FUNCTION_BLOCK FB_Startup
VAR_INPUT
END_VAR
VAR_OUTPUT
END_VAR
VAR
	timer1 : TON;
	timer2 : TON;
	timer3 : TON;
	timer4 : TON;
	timer5 : TON;
	timer6 : TON;
	timer7 : TON;
	timer14: INT;
END_VAR

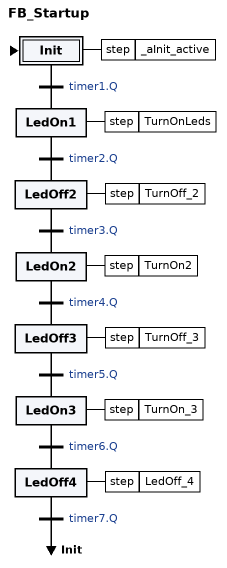
INITIAL_STEP Init:
    _aInit_active(N);  // step action
END_STEP
TRANSITION FROM Init TO LedOn1
    := timer1.Q;
END_TRANSITION
STEP LedOn1:
    TurnOnLeds(N);  // step action
END_STEP
TRANSITION FROM LedOn1 TO LedOff2
    := timer2.Q;
END_TRANSITION
STEP LedOff2:
    TurnOff_2(N);  // step action
END_STEP
TRANSITION FROM LedOff2 TO LedOn2
    := timer3.Q;
END_TRANSITION
STEP LedOn2:
    TurnOn2(N);  // step action
END_STEP
TRANSITION FROM LedOn2 TO LedOff3
    := timer4.Q;
END_TRANSITION
STEP LedOff3:
    TurnOff_3(N);  // step action
END_STEP
TRANSITION FROM LedOff3 TO LedOn3
    := timer5.Q;
END_TRANSITION
STEP LedOn3:
    TurnOn_3(N);  // step action
END_STEP
TRANSITION FROM LedOn3 TO LedOff4
    := timer6.Q;
END_TRANSITION
STEP LedOff4:
    LedOff_4(N);  // step action
END_STEP
TRANSITION FROM LedOff4 TO Init
    := timer7.Q;
END_TRANSITION

ACTION _aInit_active:
timer1(IN := TRUE, PT := T#1S);
timer2(IN := FALSE, PT := T#1S);
timer3(IN := FALSE, PT := T#1S);
timer4(IN := FALSE, PT := T#1S);
timer5(IN := FALSE, PT := T#1S);
timer6(IN := FALSE, PT := T#1S);
timer7(IN := FALSE, PT := T#1S);
AllLEDsTrigger(FALSE);
END_ACTION

METHOD AllLEDsTrigger : BOOL
VAR_INPUT
	OnOff : BOOL; // OnOff - Turn off, True - Turn On
END_VAR
GVL.LED_Comm_Fault := OnOff;
GVL.LED_EE_Grip := OnOff;
GVL.LED_EE_Ungrip := OnOff;
GVL.LED_EMG_STOP := OnOff;
GVL.LED_J1_CCW := OnOff;
GVL.LED_J1_CW := OnOff;
GVL.LED_J2_CCW := OnOff;
GVL.LED_J2_CW := OnOff;
GVL.LED_J3_CCW := OnOff;
GVL.LED_Record_Delay := OnOff;
GVL.LED_Record_Pos := OnOff;
GVL.LED_Reset := OnOff;
GVL.LED_Start_Pause := OnOff;
GVL.LED_Warning := OnOff;
END_METHOD

ACTION LedOff_4:
timer1(IN := FALSE, PT := T#1S);
timer2(IN := FALSE, PT := T#1S);
timer3(IN := FALSE, PT := T#1S);
timer4(IN := FALSE, PT := T#1S);
timer5(IN := FALSE, PT := T#1S);
timer6(IN := FALSE, PT := T#1S);
timer7(IN := TRUE, PT := T#1S);
AllLEDsTrigger(FALSE);
END_ACTION

ACTION TurnOff_2:
timer1(IN := FALSE, PT := T#1S);
timer2(IN := FALSE, PT := T#1S);
timer3(IN := TRUE, PT := T#1S);
timer4(IN := FALSE, PT := T#1S);
timer5(IN := FALSE, PT := T#1S);
timer6(IN := FALSE, PT := T#1S);
timer7(IN := FALSE, PT := T#1S);
AllLEDsTrigger(FALSE);
END_ACTION

ACTION TurnOff_3:
timer1(IN := FALSE, PT := T#1S);
timer2(IN := FALSE, PT := T#1S);
timer3(IN := FALSE, PT := T#1S);
timer4(IN := FALSE, PT := T#1S);
timer5(IN := TRUE, PT := T#1S);
timer6(IN := FALSE, PT := T#1S);
timer7(IN := FALSE, PT := T#1S);
AllLEDsTrigger(FALSE);
END_ACTION

ACTION TurnOn_3:
timer1(IN := FALSE, PT := T#1S);
timer2(IN := FALSE, PT := T#1S);
timer3(IN := FALSE, PT := T#1S);
timer4(IN := FALSE, PT := T#1S);
timer5(IN := FALSE, PT := T#1S);
timer6(IN := TRUE, PT := T#1S);
timer7(IN := FALSE, PT := T#1S);
AllLEDsTrigger(TRUE);
END_ACTION

ACTION TurnOn2:
timer1(IN := FALSE, PT := T#1S);
timer2(IN := FALSE, PT := T#1S);
timer3(IN := FALSE, PT := T#1S);
timer4(IN := TRUE, PT := T#1S);
timer5(IN := FALSE, PT := T#1S);
timer6(IN := FALSE, PT := T#1S);
timer7(IN := FALSE, PT := T#1S);
AllLEDsTrigger(TRUE);
END_ACTION

ACTION TurnOnLeds:
timer1(IN := FALSE, PT := T#1S);
timer2(IN := TRUE, PT := T#1S);
timer3(IN := FALSE, PT := T#1S);
timer4(IN := FALSE, PT := T#1S);
timer5(IN := FALSE, PT := T#1S);
timer6(IN := FALSE, PT := T#1S);
timer7(IN := FALSE, PT := T#1S);
AllLEDsTrigger(TRUE);
END_ACTION

END_FUNCTION_BLOCK

(* stored: Version 1.1.0.1, ProductVersion 3.1.4024.13
   POU FB_Startup: Id {b8621711-4300-4241-84d0-5f9d5121482f}, SpecialFunc None
   Action _aInit_active: Id {71b52ef5-6cc0-43e4-a167-2910491bd5cd}
   Method AllLEDsTrigger: Id {56fddde5-8487-4a2d-a6eb-629934013dab}
   Action LedOff_4: Id {94ed513a-ae2b-4cde-903b-69a55d112c27}
   Action TurnOff_2: Id {c59e4578-f57a-4218-9698-0c1ab6dfa985}
   Action TurnOff_3: Id {57fbf166-0860-45ab-be27-5cce5f0cc7ef}
   Action TurnOn_3: Id {1550c02f-8f01-4518-a7ac-da0652c13590}
   Action TurnOn2: Id {2d094cb6-ab78-469e-8c8d-63a456ac6d88}
   Action TurnOnLeds: Id {9770b222-a122-43ae-9df8-13ef0f886ac4} *)
